Fanuc KAREL source: kd00032.KL

-- PROVISIONAL review KL for V770-1; original PC SHA256 fc813401e89ed233813f3bbaf5a49ee5a7b807595c7369281c018090ecc2f442
-- Incomplete behavior may be omitted. Consult companion uncertainty JSON. Do not deploy.
PROGRAM KD00032
%NOLOCKGROUP
VAR
  I : INTEGER
  J : INTEGER
  B : BOOLEAN
  R : REAL
  S : STRING[80]
BEGIN
  -- UNRESOLVED_PC offsets 5-25; opcodes 9D,81,18,2E,12,22,9D,13,04
  -- UNRESOLVED_PC offsets 30-34; opcodes 7F
END KD00032
